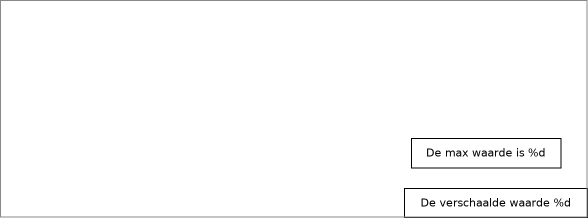
VISUALIZATION Visualization  // 588x218
    Rectangle (411,138 150x30), "De max waarde is %d", text variable: MAIN.nScaledMax
        OnMouseDown: write the text variable via Default
    Rectangle (404,188 184x30), "De verschaalde waarde %d", text variable: MAIN.Waarde
END_VISUALIZATION

(* stored: Version 1.1.0.1, ProductVersion 3.1.4024.12
   Visu Visualization: Id {aed89d90-7be6-4e24-8c83-7d6df98885fe} *)
